// TIA Portal V20 export
DATA_BLOCK "SP503"   // DB319
// stored: MemoryReserve 100
   VAR
      "UPPER 2-1 HEATER TEMPERATURE CONTROLLER ALARM" : Bool;
      SPARE : Bool;
      "UPPER 2-2 HEATER TEMPERATURE CONTROLLER ALARM" : Bool;
      SPARE_1 : Bool;
      "LOWER 2-1 HEATER TEMPERATURE CONTROLLER ALARM" : Bool;
      SPARE_2 : Bool;
      "LOWER 2-2 HEATER TEMPERATURE CONTROLLER ALARM" : Bool;
      SPARE_3 : Bool;
      "LOWER 2-3 HEATER TEMPERATURE CONTROLLER ALARM" : Bool;
      SPARE_4 : Bool;
      SPARE_5 : Bool;
      SPARE_6 : Bool;
      SPARE_7 : Bool;
      SPARE_8 : Bool;
      "STACK-1 LIGHT CURTAIN STATUS/SELECT" : Bool;
      "STACK-2 LIGHT CURTAIN STATUS/SELECT" : Bool;
   END_VAR
BEGIN
END_DATA_BLOCK
